TYPE E_MachineState :
(
    Idle,
    Running,
    Filling,
    Capping,
    Stopped

);
END_TYPE

(* stored: Version 1.1.0.1, ProductVersion 3.1.4024.16
   DUT E_MachineState: Id {eeef3a60-161b-4078-a769-884402a4f528} *)
